KUKA KRL data list: AtualizaVariaveis.dat

&ACCESS RV
DEFDAT AtualizaVariaveis

ENDDAT
